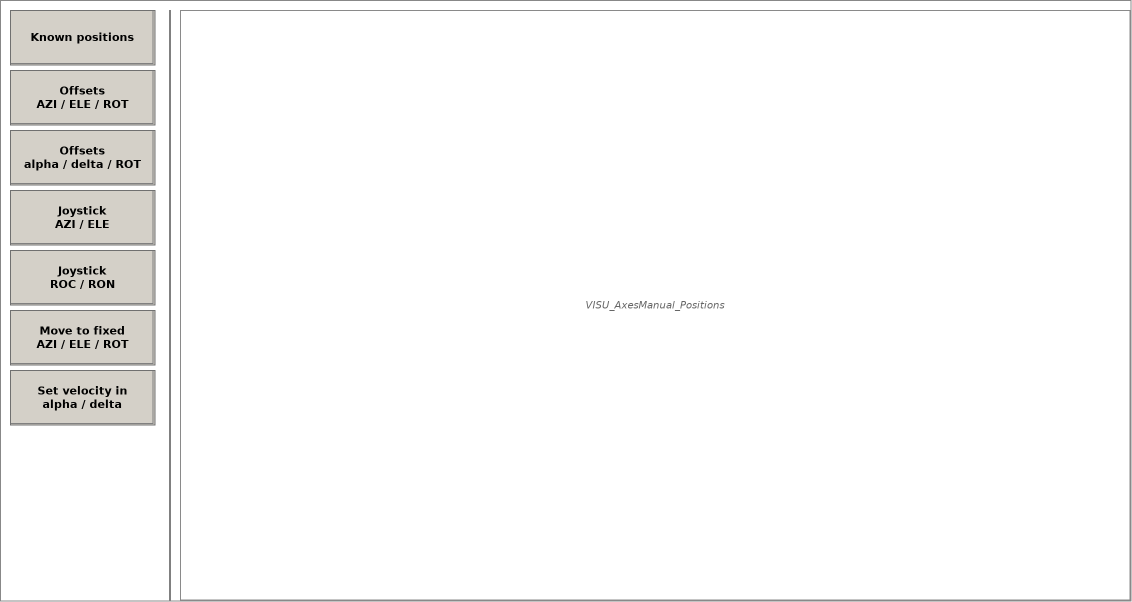
VISUALIZATION VISU_AxesManual  // 1132x602
VAR_IN_OUT
	ref : Axes;
    widget : AxesManualWidget;
END_VAR
    Button (10,10 145x55), "Known positions", pressed state: widget.activeTab = AxesManualTabs.TAB_POSITIONS
        OnMouseClick: execute { widget.activeTab := AxesManualTabs.TAB_POSITIONS; }
    Button (10,190 145x55), "Joystick AZI / ELE", pressed state: widget.activeTab = AxesManualTabs.TAB_JOYSTICK_AZIELE
        OnMouseClick: execute { widget.activeTab := AxesManualTabs.TAB_JOYSTICK_AZIELE; }
    Button (10,250 145x55), "Joystick ROC / RON", pressed state: widget.activeTab = AxesManualTabs.TAB_JOYSTICK_ROT
        OnMouseClick: execute { widget.activeTab := AxesManualTabs.TAB_JOYSTICK_ROT; }
    Button (10,70 145x55), "Offsets AZI / ELE / ROT", pressed state: widget.activeTab = AxesManualTabs.TAB_OFFSETS_AZIELE
        OnMouseClick: execute { widget.activeTab := AxesManualTabs.TAB_OFFSETS_AZIELE; }
    Button (10,310 145x55), "Move to fixed AZI / ELE / ROT", pressed state: widget.activeTab = AxesManualTabs.TAB_MOVEABSOLUTE
        OnMouseClick: execute { widget.activeTab := AxesManualTabs.TAB_MOVEABSOLUTE; }
    Button (10,370 145x55), "Set velocity in alpha / delta", pressed state: widget.activeTab = AxesManualTabs.TAB_MOVEVELOCITY
        OnMouseClick: execute { widget.activeTab := AxesManualTabs.TAB_MOVEVELOCITY; }
    Line (170,600) (170,10)
    Frame (180,10 950x590), frame switch variable: widget.activeTab
        shows VISU_AxesManual_Positions(ref := ref, widget := widget.positions)
        shows VISU_AxesManual_Joystick_AziEle(ref := ref, widget := widget.joystickAziEle)
        shows VISU_AxesManual_Joystick_Rot(ref := ref, widget := widget.joystickRot)
        shows VISU_AxesManual_Offsets_AziEleRot(ref := ref, widget := widget.offsets)
        shows VISU_AxesManual_Offsets_AlphaDeltaRot(ref := ref, widget := widget.offsets)
        shows VISU_AxesManual_MoveAbsolute(ref := ref, widget := widget.moveAbsolute)
        shows VISU_AxesManual_MoveVelocity(ref := ref, widget := widget.moveVelocity)
    Button (10,130 145x55), "Offsets alpha / delta / ROT", pressed state: widget.activeTab = AxesManualTabs.TAB_OFFSETS_ALPHADELTA
        OnMouseClick: execute { widget.activeTab := AxesManualTabs.TAB_OFFSETS_ALPHADELTA; }
END_VISUALIZATION

(* stored: Version 1.1.0.1, ProductVersion 3.1.4019.2
   Visu VISU_AxesManual: Id {0b83c5b4-db47-4d0d-891b-5d638822c6dd} *)
